FUNCTION_BLOCK PUBLIC FB_AirConditioning
VAR_OUTPUT
	bActive			: BOOL;
	lrTemperature	: LREAL;
END_VAR

METHOD PUBLIC Activate
bActive := TRUE;
END_METHOD

PROPERTY PUBLIC Activated : BOOL
GET
Activated := bActive;
END_GET
END_PROPERTY

METHOD PUBLIC Deactivate
bActive := false;
END_METHOD

METHOD PUBLIC SetTemperature : BOOL
VAR_INPUT
	lrNewTemperature	:	LREAL;
END_VAR
lrTemperature := lrNewTemperature;
END_METHOD

PROPERTY PUBLIC Temperature : LREAL
GET
Temperature := lrTemperature;
END_GET
END_PROPERTY

END_FUNCTION_BLOCK

(* stored: Version 1.1.0.1, ProductVersion 3.1.4024.12
   POU FB_AirConditioning: Id {8e25d5ec-9a86-4a82-9baf-9098ed0aab4d}, SpecialFunc None
   Method Activate: Id {d1feb8e2-e998-44dc-b637-5e9a76d6afe5}
   Property Activated: Id {ce726444-f01f-4c74-94e8-5b017ae6a034}
   Get Get: Id {d192b8ef-675e-4964-a89b-57fd2dcef6e7}
   Method Deactivate: Id {7f6cdbb9-87ab-4e54-9cd3-e8c9e571dfae}
   Method SetTemperature: Id {22060a4c-cb7f-4541-90fb-013901bc3836}
   Property Temperature: Id {f8152be3-3bb2-4a2f-b79b-8d1426ba408f}
   Get Get: Id {79d47eb5-b67c-4a99-b6b6-1eaf7b168feb} *)
